Omron Sysmac Studio project PLC Project_1 (Sysmac Studio 1.58.0.9, StandardProject)

# Controller PLC: NX102-1000 version 1.50
Units and slaves: Unit 1 : NX-PF0730 (N1)
Task PrimaryTask (priority 4, period or condition 2000): Program1

TYPE dt_Settings : STRUCT
    colourFilter : ColourFilter;
    filter_1 : UINT;
    filter_2 : UINT;
    frame_cutout : MaxMin;
    lines : UINT;
    cam_settings : CamSettings;
END_STRUCT END_TYPE
TYPE MaxMin : STRUCT
    Max : UINT;
    Min : UINT;
END_STRUCT END_TYPE
TYPE ColourFilter : STRUCT
    hue : MaxMin;
    saturation : MaxMin;
    value : MaxMin;
END_STRUCT END_TYPE
TYPE MESSAGETYPE : (LINE_VALUE := 0, SETTING := 1, ALIVE := 2, REQUEST_SETTINGS := 3, IDLE := 4, PLC_CONFIRM := 5); END_TYPE
TYPE CamSettings : STRUCT
    ReverseX : BOOL;
    ReverseY : BOOL;
    ExposureTime : REAL;
    ColorTransformationEnable : BOOL;
END_STRUCT END_TYPE

VAR_GLOBAL
    line_values : ARRAY[0..19] OF BYTE;
END_VAR

PROGRAM Program1
VAR
    OpenServer : SktTCPAccept;
    ReceiveData : SktTCPRcv;
    SendData : SktTCPSend;
    Socket : _sSOCKET;
    RcvDat : ARRAY[0..1999] OF BYTE;
    SendDat : ARRAY[0..1999] OF BYTE;
    SendDataSize : UINT;
END_VAR
VAR RETAIN
    settings : dt_Settings;
END_VAR
VAR
    CloseSocket : SktClose;
    unknown_command_received : UINT;
    line_values_received_counter : UINT;
    receivedCommand : MESSAGETYPE;
    sendCommand : MESSAGETYPE;
    ReceivedDataSize : UINT;
    settingsSendCounter : UINT;
    requestSettingsCounter : UINT;
    receivedCounter : UINT;
    RetriggerOpenServer : TON;
    retriggerCounter : UINT;
    settingsHaveChanged : BOOL;
    ReceivedDoneLastCycle : BOOL;
    settingsReceivedCounter : UINT;
    CycleCounter : UINT;
    CyclesBetweenEachSend : UINT;
    MilisecondsBetweenEachFrameUpdate : UINT;
    SettingsAsByte : ARRAY[0..1999] OF BYTE;
    DataStructLength : UINT;
    Gewicht : LREAL;
    StrData : STRING[1890];
    Value : LREAL;
    x : UINT;
END_VAR
VAR_EXTERNAL
    line_values : ARRAY[0..19] OF BYTE;
END_VAR
//-----------------------------------------------------------------------------------------------------------
//---------------------------------BASIC TCP SOCKET COMMUNICATION------------------------------------
//-----------------------------------------------------------------------------------------------------------

//Open a TCP-Socket Server
OpenServer.Execute := 	NOT OpenServer.Execute
										OR OpenServer.Done
										OR OpenServer.Busy;
RetriggerOpenServer(	In:=OpenServer.Busy
									AND NOT OpenServer.Done
									AND OpenServer.Execute, PT:=t#5s);

IF CloseSocket.Busy THEN OpenServer.Execute := FALSE; END_IF;
//IF RetriggerOpenServer.Q THEN OpenServer.Execute := FALSE; Inc(retriggerCounter); END_IF;

OpenServer(Execute:=OpenServer.Execute, SrcTcpPort:=2100, TimeOut:=50, Socket=>Socket);

//If the client is connected start to listen. Retrigger this command everytime a Response has been send
ReceiveData.Execute := OpenServer.Done AND NOT SendData.Done;
ReceiveData(	Execute:=ReceiveData.Execute,
						Socket:=Socket,
						TimeOut:=50,
						Size:=2000,
						RcvDat:=RcvDat[0]);

//Send Response after receiving data
SendData.Execute := ReceiveData.Done;
SendData(	Execute:=ReceiveData.Done,
		 			Socket:=Socket,
					SendDat:=SendDat[0],
					Size:=SendDataSize);

//Close the Socket on error
CloseSocket.Execute := (OpenServer.Error
										OR ReceiveData.Error
										OR SendData.Error
										OR RetriggerOpenServer.Q)
										AND NOT CloseSocket.Execute
										OR CloseSocket.Busy	;
CloseSocket(	Execute:=CloseSocket.Execute, Socket:=Socket);


//-----------------------------------------------------------------------------------------------------------
//---------------------------------LOGIC FOR RECEIVING AND SENDING DATA-------------------------
//-----------------------------------------------------------------------------------------------------------

IF ReceiveData.Done  AND NOT ReceivedDoneLastCycle THEN
	Inc(receivedCounter);
	ReceivedDataSize := ReceiveData.RcvSize;
	
	NumToEnum(	BYTE_TO_DINT(RcvDat[0]),
			  				receivedCommand);
	CASE receivedCommand OF
		IDLE:
			sendCommand := PLC_CONFIRM;
	    LINE_VALUE:
			MemCopy(	In:=RcvDat[1],
								AryOut:=line_values[0],
								Size:=20);
			sendCommand := PLC_CONFIRM;
			Inc(line_values_received_counter);
			
		SETTING:
			AryByteTo(	In:=RcvDat[1],
					  			Size:=ReceivedDataSize-1,
					  			Order:=_eBYTE_ORDER#_LOW_HIGH,
								OutVal:=settings);
			sendCommand := PLC_CONFIRM;
			Inc(settingsReceivedCounter);
		 REQUEST_SETTINGS:
			sendCommand := SETTING;
			Inc(requestSettingsCounter);
	ELSE
		sendCommand := PLC_CONFIRM;
	   	Inc(unknown_command_received);
	END_CASE;
	
	IF sendCommand = PLC_CONFIRM THEN
		IF settingsHaveChanged THEN
			sendCommand := SETTING;
			settingsHaveChanged := FALSE;
		END_IF;
	END_IF;
	
	SendDat[0] := DINT_TO_BYTE(EnumToNum(sendCommand));
	CASE sendCommand OF
		SETTING:
			SendDataSize := 1 + ToAryByte(	In:=settings,
					  											Order:=_eBYTE_ORDER#_LOW_HIGH,
																AryOut:=SendDat[1]);
			Inc(settingsSendCounter);
	ELSE
		//PLC_CONFIRM:
		SendDataSize := 1;
	END_CASE;
END_IF;


//-----------------------------------------------------------------------------------------------------------
//---------------------------------DEBUG STUFF-----------------------------------------------------------
//-----------------------------------------------------------------------------------------------------------

INC(CycleCounter);
IF ReceivedDoneLastCycle <> ReceiveData.Done AND ReceiveData.Done THEN
	MilisecondsBetweenEachFrameUpdate := CycleCounter * LINT_TO_UINT(TimeToNanoSec(GetMyTaskInterval()) / 1000000);
	CycleCounter := 0;
END_IF;

ReceivedDoneLastCycle := ReceiveData.Done;

DataStructLength := ToAryByte(	In:=settings,
					Order:=_eBYTE_ORDER#_LOW_HIGH,
					AryOut:=SettingsAsByte[0]);


		
END_PROGRAM

# Device HMI (NA): not converted